INTERFACE ITF_BaseHMITopElement_Command EXTENDS ITF_BaseHMIGroupElement_Command

END_INTERFACE

(* stored: Version 1.1.0.1
   Itf ITF_BaseHMITopElement_Command: Id {6900ea0f-d4e3-0307-2f75-efdf9ef303ef} *)
